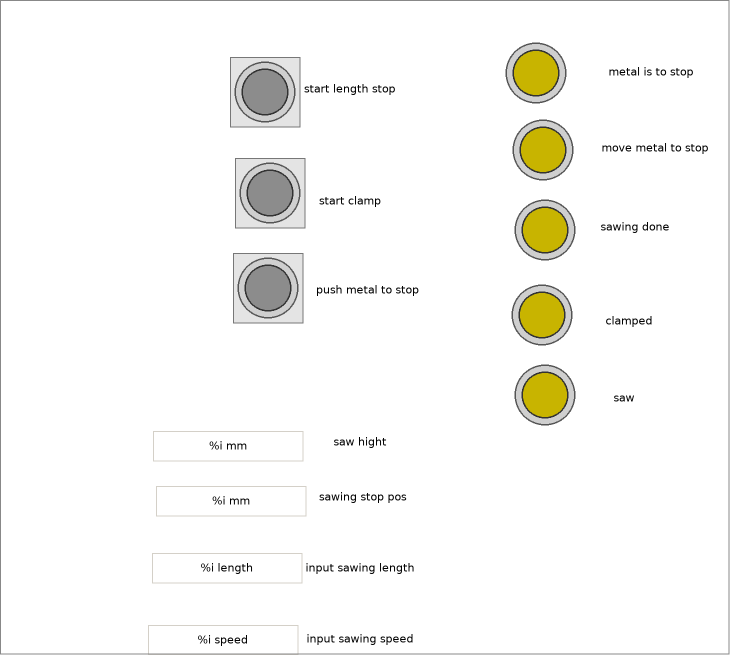
VISUALIZATION Visualization_1  // 730x655
    PushSwitch (230,57 70x70), variable: POU_UserInterface.startButtonLengthStop, behaviour: TOGGLE, style: Switch-PushSwitch-Gray
    Lamp1 (508,115 70x70), variable: POU_UserInterface.messageMoveMetalToStop, style: Lamp-Lamp1-Yellow
    Lamp1 (510,195 70x70), variable: POU_UserInterface.sawingDone, style: Lamp-Lamp1-Yellow
    Textfield (152,553 150x30), "%i length", text variable: POU_UserInterface.inputSawingLength
        OnMouseClick: write the text variable via Default
    Textfield (148,625 150x30), "%i speed", text variable: POU_UserInterface.inputSawingSpeed
        OnMouseClick: write the text variable via Default
    Label (580,133 150x30), "move metal to stop"
    Label (560,212 150x30), "sawing done"
    Label (275,186 150x30), "start clamp"
    Label (288,482 150x30), "sawing stop pos"
    Label (275,74 150x30), "start length stop"
    Label (285,624 150x30), "input sawing speed"
    Textfield (156,486 150x30), "%i mm", text variable: POU_SawLengthStop.sawingStopPos
    Label (285,553 150x30), "input sawing length"
    PushSwitch (233,253 70x70), variable: POU_SawLengthStop.metalAgainstStop, behaviour: TOGGLE, style: Switch-PushSwitch-Gray
    Label (292,275 151x30), "push metal to stop"
    Lamp1 (501,38 70x70), variable: POU_UserInterface.signStartClamping, style: Lamp-Lamp1-Yellow
    Label (578,57 150x30), "metal is to stop"
    PushSwitch (235,158 70x70), variable: POU_UserInterface.startClamp, behaviour: TOGGLE, style: Switch-PushSwitch-Gray
    Label (285,427 150x30), "saw hight"
    Textfield (153,431 150x30), "%i mm", text variable: POU_Saw.actualPos
    Lamp1 (507,280 70x70), variable: POU_Clamp.clampingDone, style: Lamp-Lamp1-Yellow
    Label (554,306 150x30), "clamped"
    Lamp1 (510,360 70x70), variable: POU_Saw.saw, style: Lamp-Lamp1-Yellow
    Label (549,383 150x30), "saw"
END_VISUALIZATION

(* stored: Version 1.1.0.1, ProductVersion 3.1.4024.12
   Visu Visualization_1: Id {b767637b-73f3-43cc-8e82-5650a0d8700a} *)
